{attribute addProperty BoxType "EL2502-0010-0020"}
{attribute addProperty Id "PWM_Inputs_Channel_1AT %I*PWM_Inputs_Channel_F0CD9CDB1620PWM_SysTime_Channel_1AT %I*PWM_SysTime_Channel_D079C8006480PWM_Per_DC_Outputs_Channel_1AT %Q*PWM_Per_DC_Outputs_Channel_93D6009A112140WcStateAT %I*WcState_F855686C1620InfoDataAT %I*InfoData_BC63D37F80100"}
{attribute addProperty CRC "1832466045"}
{attribute addProperty SizeInBites "288"}
{attribute addProperty SizeInBytes "36"}
TYPE EL2502_746480DE :
STRUCT
	{attribute addProperty Name "PWM_Inputs_Channel_1"}
	PWM_Inputs_Channel_1 : PWM_Inputs_Channel_F0CD9CDB;
	{attribute addProperty Name "PWM_SysTime_Channel_1"}
	PWM_SysTime_Channel_1 : PWM_SysTime_Channel_D079C800;
	{attribute addProperty Name "PWM_Per_DC_Outputs_Channel_1"}
	PWM_Per_DC_Outputs_Channel_1 : PWM_Per_DC_Outputs_Channel_93D6009A;
	{attribute addProperty Name "WcState"}
	WcState : WcState_F855686C;
	{attribute addProperty Name "InfoData"}
	InfoData : InfoData_BC63D37F;
END_STRUCT
END_TYPE

(* stored: Version 1.2.0.0, ProductVersion 3.1.4024.9
   DUT EL2502_746480DE: Id {d614a33d-8394-464e-bfeb-fc061eb5ec89} *)
